// TwinCAT 3 PLC project PowerMonitoringSample
// ProgramVersion: 3.1.4022.3
// libraries:
//   Tc2_Standard, * (Beckhoff Automation GmbH)
//   Tc2_System, * (Beckhoff Automation GmbH)
//   Tc2_Utilities, * (Beckhoff Automation GmbH)
//   Tc3_EventLogger, * (Beckhoff Automation GmbH)
//   Tc3_Module, * (Beckhoff Automation GmbH)
//   Tc3_PowerMonitoring, * (Beckhoff Automation GmbH)
// project tree:
//   DUTs/ E_AnalysisIDs.TcDUT, ST_EL3783_InputSamples.TcDUT, ST_EL3783_InputSamples_Scaled.TcDUT
//   GVLs/ Global_Constants.TcGVL
//   / PlcTask.TcTTO, PlcTaskSlow.TcTTO
//   POUs/ DateTimeClock.TcPOU, MAIN.TcPOU, MAIN_SLOW.TcPOU
//   POUs/TestSignalGeneration/ FB_GenerateInputSignal_1Ph.TcPOU
//   POUs/TestSignalGeneration/SignalGeneration/ E_FunctionType.TcDUT, FB_FunctionGenerator_plusPhi.TcPOU

CONFIGURATION PowerMonitoringSample
    RESOURCE PLC ON TwinCAT3
        TASK PlcTask(INTERVAL := T#1ms, PRIORITY := 4);
        TASK PlcTaskSlow(INTERVAL := T#10ms, PRIORITY := 8);
        PROGRAM MAIN WITH PlcTask : MAIN;
        PROGRAM MAIN_SLOW WITH PlcTaskSlow : MAIN_SLOW;
    END_RESOURCE
END_CONFIGURATION

// ---- DUTs/E_AnalysisIDs.TcDUT
{attribute 'qualified_only'}
{attribute 'strict'}
TYPE E_AnalysisIDs :
(
(* analysis chain TimeBased *)
	 Source_TimeBased :=1,
	 Frequency_TimeBased,
	 BasicValues_TimeBased,
	 PowerValues_TimeBased,
(* analysis chain FrequencyBased *)	
	Source_FrequencyBased,
	PowerValues_FrequencyBased,
	Spectrum_FrequencyBased,
	Harmonics_FrequencyBased	
) UDINT;
END_TYPE

// ---- DUTs/ST_EL3783_InputSamples.TcDUT
TYPE ST_EL3783_InputSamples :
STRUCT
(* Inputs from EL3783 *)
	aUL1		: ARRAY[1..cOversamples] OF INT;
	aUL2		: ARRAY[1..cOversamples] OF INT;
	aUL3		: ARRAY[1..cOversamples] OF INT;
	aIL1		: ARRAY[1..cOversamples] OF INT;
	aIL2		: ARRAY[1..cOversamples] OF INT;
	aIL3		: ARRAY[1..cOversamples] OF INT;
END_STRUCT
END_TYPE

// ---- DUTs/ST_EL3783_InputSamples_Scaled.TcDUT
TYPE ST_EL3783_InputSamples_Scaled :
STRUCT
(* Inputs from EL3783 *)
	aUL1		: ARRAY[1..cOversamples] OF LREAL;
	aUL2		: ARRAY[1..cOversamples] OF LREAL;
	aUL3		: ARRAY[1..cOversamples] OF LREAL;
	aIL1		: ARRAY[1..cOversamples] OF LREAL;
	aIL2		: ARRAY[1..cOversamples] OF LREAL;
	aIL3		: ARRAY[1..cOversamples] OF LREAL;
END_STRUCT
END_TYPE

// ---- POUs/TestSignalGeneration/SignalGeneration/E_FunctionType.TcDUT
TYPE E_FunctionType :
(
	eSine,
	eSquare,
	ePulse,
	eTriangular,
	eSawtooth,	
	eAM
);
END_TYPE

// ---- GVLs/Global_Constants.TcGVL
VAR_GLOBAL CONSTANT
	cOversamples			: UDINT := 10;
	cSamplerate				: UDINT := 10_000;
(*
	cFFTLength				: UDINT := 2048;
	cWindowLength			: UDINT := 1600;	
*)	
	cFFTLength				: UDINT := 4096;
	cWindowLength			: UDINT := 3200;

	cBufferLength			: UDINT := cWindowLength/2;
	
	cHarmonicBands			: UDINT := 20;
	cNumQuantiles			: UDINT := 2;
	cFreqMode				: LREAL := 50.0;
END_VAR

// ---- POUs/MAIN.TcPOU
PROGRAM MAIN
VAR CONSTANT
(* Init parameters*)
	cSourceTimeBasedInitPars		: ST_PMA_Source_InitPars 		   		:= (nBufferLength := cOversamples);	
	cSourceFrequencyBasedInitPars	: ST_PMA_Source_InitPars 		   		:= (nBufferLength := cBufferLength);

	cFrequencyInitPars				: ST_PMA_Frequency_Period_InitPars 		:= (nBufferLength := cOversamples, fSampleRate := cSamplerate, fMinFreq := 40, fMaxFreq := 70, nPeriods := 1, nFilterOrder := 2, fCutoff := 70, eInputSelect := E_PMA_InputSelect.Voltage, fMinInput := 150);
	cBasicValuesInitPars			: ST_PMA_BasicValues_Period_InitPars 	:= (nBufferLength := cOversamples, fSampleRate := cSamplerate, fMinInputCurrent := 0.1);
	cPowerValuesInitPars			: ST_PMA_PowerValues_Period_InitPars 	:= (nBufferLength := cOversamples, fSampleRate := cSamplerate, fMinInputCurrent := 0.1);
	cScalingEL3783Pars				: ST_PMA_Scaling_EL3783_InitPars 	 	:= (nOversamples  := cOversamples, fOffsetVoltage := 0, fGainVoltage := 1, fOffsetCurrent := 0, fGainCurrent := 1, fFactorCurrentTransformer := 1);													
END_VAR
VAR	
(* Inputs*)
	nInputSelect				: INT := 1; 						// 1: generate signal, 2: input EL3783
	stEL3783_1_In 				AT%I* : ST_EL3783_InputSamples;
	stEL3783_1_Scaled			: ST_EL3783_InputSamples_Scaled;
	bEL3783_HcRangeActive 		AT%I* : BOOL;
	aEL3783_HcRange 			AT%I* : ARRAY [0..3] OF USINT;	
	
	fbGenerateInputs			: FB_GenerateInputSignal_1Ph;									
	fSetPhaseDiff				: LREAL := 5;	
	fFreqSetpoint				: LREAL	:= 50;
	fAmplitudeVoltage			: LREAL	:= 230*SQRT(2);
	fAmplitudeCurrent			: LREAL	:= 1*SQRT(2);
	bEnableHarmonics			: BOOL	:= FALSE;

(* Functionblocks *)
	fbScaling					: FB_PMA_Scaling_EL3783 		:= (stInitPars:= cScalingEL3783Pars);
	fbSource_TimeBased			: FB_PMA_Source_1Ph 			:= (nOwnID:= E_AnalysisIDs.Source_TimeBased, 		aDestIDs:= [E_AnalysisIDs.Frequency_TimeBased, E_AnalysisIDs.BasicValues_TimeBased, E_AnalysisIDs.PowerValues_TimeBased], stInitPars:= cSourceTimeBasedInitPars);
	fbSource_FrequencyBased		: FB_PMA_Source_1Ph				:= (nOwnID:= E_AnalysisIDs.Source_FrequencyBased, 	aDestIDs:= [E_AnalysisIDs.PowerValues_FrequencyBased, E_AnalysisIDs.Spectrum_FrequencyBased, E_AnalysisIDs.Harmonics_FrequencyBased], stInitPars:= cSourceFrequencyBasedInitPars);
	fbFrequency					: FB_PMA_Frequency_Period_1Ph 	:= (nOwnID:= E_AnalysisIDs.Frequency_TimeBased, 	stInitPars:= cFrequencyInitPars);
	fbBasicValues				: FB_PMA_BasicValues_Period_1Ph := (nOwnID:= E_AnalysisIDs.BasicValues_TimeBased, 	stInitPars:= cBasicValuesInitPars);
	fbPowerValues				: FB_PMA_PowerValues_Period_1Ph := (nOwnID:= E_AnalysisIDs.PowerValues_TimeBased, 	stInitPars:= cPowerValuesInitPars);
		
(* Control *)
	bResetStatistics			: BOOL;	
	
// Errorhandling
	bError						: BOOL;
	nCountErrors				: UDINT;
	nEventId					: UDINT;
	sEventClassName				: T_MaxString;
	sSourcePath					: T_MaxString;
	eSeverity					: TcEventSeverity;
	ipResultMessage				: I_TcMessage;
	
//Liam's variable for TcHmi
	bResetEnergyRecord : BOOL:= FALSE;
	
END_VAR

bError := FALSE;

(**************************************************************************************************************)
(* Inputs *)
CASE nInputSelect OF
	1:	(* signal generation from PLC *)
		fbGenerateInputs.Call(	bEnableHarmonics			:= bEnableHarmonics,
								fSetFrequency				:= fFreqSetpoint,		// Hz
								fSetAmplitudeVoltage		:= fAmplitudeVoltage,	// peak amplitude of sin signal
								fSetAmplitudeCurrent		:= fAmplitudeCurrent,
								fSetPhasedifferenceCurrent	:= fSetPhaseDiff,
								stEL3783_Scaled				=> stEL3783_1_Scaled);										

	2:	(* signal from terminal *)
		InputEL3783();
		IF fbScaling.bError THEN
			bError := TRUE;
			ipResultMessage := fbScaling.ipResultMessage;
		END_IF
END_CASE

(**************************************************************************************************************)
(* Source *)
fbSource_TimeBased.Call(pBuffer_U:= ADR(stEL3783_1_Scaled.aUL1),			 
						pBuffer_I:= ADR(stEL3783_1_Scaled.aIL1),
						nDataInSizePerCh:= SIZEOF(stEL3783_1_Scaled)/6, // Caused by 3Ph Buffer!
						nOptionPars:= 0);
IF fbSource_TimeBased.bError THEN
	bError := TRUE;
	ipResultMessage := fbSource_TimeBased.ipResultMessage;
END_IF
	
fbSource_FrequencyBased.Call(pBuffer_U:= ADR(stEL3783_1_Scaled.aUL1),			 
							 pBuffer_I:= ADR(stEL3783_1_Scaled.aIL1),		
							 nDataInSizePerCh:= SIZEOF(stEL3783_1_Scaled)/6, // Caused by 3Ph Buffer!
							 nOptionPars:= 0);
IF fbSource_FrequencyBased.bError THEN
	bError := TRUE;
	ipResultMessage := fbSource_FrequencyBased.ipResultMessage;
END_IF
				
(**************************************************************************************************************)
(* Algorithms *)

(* Frequency *)
IF NOT fbFrequency.Call(bResetStatistics:= bResetStatistics) THEN
	bError := TRUE;
	ipResultMessage := fbFrequency.ipResultMessage;	
END_IF

(* Basic Values *)
IF NOT fbBasicValues.Call(fFreq:= fbFrequency.fFreq, bResetStatistics:= bResetStatistics) THEN
	bError := TRUE;
	ipResultMessage := fbBasicValues.ipResultMessage;
END_IF

(* Power Values *)

(*Liam's Code for TcHmi control and Monitor*)
//Thêm biến bResetEnergyRecord vào để điều khiển quá trình reset lại giá trị của kWh
IF NOT fbPowerValues.Call(fFreq:= fbFrequency.fFreq, bResetEnergyCalc := bResetEnergyRecord, bResetStatistics:= bResetStatistics) THEN
	bError := TRUE;
	ipResultMessage := fbPowerValues.ipResultMessage;
END_IF

(**************************************************************************************************************)
(* Event reporting *)
IF ipResultMessage <> 0 THEN	
	nEventId 		:= ipResultMessage.nEventId;
	sSourcePath 	:= ipResultMessage.ipSourceInfo.sName;
	eSeverity 		:= ipResultMessage.eSeverity;
	
	ipResultMessage.RequestEventClassName(1033, sEventClassName, SIZEOF(sEventClassName));
END_IF
IF bError THEN
	nCountErrors := nCountErrors + 1;
END_IF


(*Liam's Code for TcHmi control and Monitor*)
DateTimeClock();

ACTION InputEL3783:
(* //Autorange
fbScaling.Call_1Ph_Autorange(	pInputBuffer_U			:= ADR(stEL3783_1_In.aUL1), 
								pInputBuffer_I			:= ADR(stEL3783_1_In.aIL1), 
								nInputBufferSize		:= SIZEOF(stEL3783_1_In)/6, 
								pOutputBuffer_U			:= ADR(stEL3783_1_Scaled.aUL1), 
								pOutputBuffer_I			:= ADR(stEL3783_1_Scaled.aIL1), 
								nOutputBufferSize		:= SIZEOF(stEL3783_1_Scaled)/6, 
								bEL3783_HcRangeActive	:= bEL3783_HcRangeActive, 
								aEL3783_HcRange			:= aEL3783_HcRange);

*)		
fbScaling.Call_1Ph(	pInputBuffer_U		:= ADR(stEL3783_1_In.aUL1), 
					pInputBuffer_I		:= ADR(stEL3783_1_In.aIL1), 
					nInputBufferSize	:= SIZEOF(stEL3783_1_In)/6, 
					pOutputBuffer_U		:= ADR(stEL3783_1_Scaled.aUL1), 
					pOutputBuffer_I		:= ADR(stEL3783_1_Scaled.aIL1), 
					nOutputBufferSize	:= SIZEOF(stEL3783_1_Scaled)/6,
					bUse_5A_Range		:= FALSE);
END_ACTION

END_PROGRAM

// ---- POUs/TestSignalGeneration/FB_GenerateInputSignal_1Ph.TcPOU
FUNCTION_BLOCK FB_GenerateInputSignal_1Ph
VAR_INPUT
	fSetFrequency						: LREAL:= 50;		// Hz
	fSetAmplitudeVoltage				: LREAL:= 325;		// peak amplitude of sin signal	
	fSetAmplitudeCurrent				: LREAL:= 2;		// peak amplitude of sin signal	
	fSetPhasedifferenceCurrent			: LREAL:= 0;
END_VAR
VAR_OUTPUT
END_VAR
VAR
	fbFunctionGeneratorVoltage_L1_1		: FB_FunctionGenerator_plusPhi;	// Signal generation
	fbFunctionGeneratorVoltage_L1_2		: FB_FunctionGenerator_plusPhi;	// Signal generation
	fbFunctionGeneratorCurrent_L1		: FB_FunctionGenerator_plusPhi;	// Signal generation
	fbFunctionGeneratorCurrent_L1_2		: FB_FunctionGenerator_plusPhi;	// Signal generation
	fbFunctionGeneratorCurrent_L1_3		: FB_FunctionGenerator_plusPhi;	// Signal generation

	aBufferGen_VoltageL1_1				: ARRAY[1..cOversamples] OF LREAL;
	aBufferGen_VoltageL1_2				: ARRAY[1..cOversamples] OF LREAL;
	aBufferGen_CurrentL1_1				: ARRAY[1..cOversamples] OF LREAL;
	aBufferGen_CurrentL1_2				: ARRAY[1..cOversamples] OF LREAL;
	aBufferGen_CurrentL1_3				: ARRAY[1..cOversamples] OF LREAL;
END_VAR

METHOD Call
VAR CONSTANT
	cHarm_U_FreqFactor					: LREAL	:= 20.0; // 20th harmonic
	cHarm_U_AmpFactor					: LREAL	:= 0.1;//0.10;
	
	cHarm_I_FreqFactor_1				: LREAL	:= 7.0;
	cHarm_I_AmpFactor_1					: LREAL	:= 0.015;//0.15;
	cHarm_I_FreqFactor_2				: LREAL	:= 20.0;
	cHarm_I_AmpFactor_2					: LREAL	:= 0.01;//0.10;
END_VAR
VAR_INPUT
	bEnableHarmonics					: BOOL	:= FALSE;
	fSetFrequency						: LREAL	:= 50;		// Hz
	fSetAmplitudeVoltage				: LREAL	:= 325;		// peak amplitude of sin signal	
	fSetAmplitudeCurrent				: LREAL	:= 2;		// peak amplitude of sin signal	
	fSetPhasedifferenceCurrent			: LREAL	:= 0;
END_VAR
VAR_OUTPUT
	stEL3783_Scaled						: ST_EL3783_InputSamples_Scaled;
END_VAR
VAR
	i									: UDINT;
END_VAR
(* signal generator *)		
// L1
fbFunctionGeneratorVoltage_L1_1(fFrequency 	:= fSetFrequency,							// "Voltage - 1st harmonic"
								fAmplitude 	:= fSetAmplitudeVoltage,
								fPhi		:= 0,
								eFunction 	:= E_FunctionType.eSine,
								aSignal		:= aBufferGen_VoltageL1_1);		

fbFunctionGeneratorVoltage_L1_2(fFrequency 	:= fSetFrequency*cHarm_U_FreqFactor,		// "Voltage - harmonic"
								fAmplitude 	:= fSetAmplitudeVoltage*cHarm_U_AmpFactor,
								fPhi		:= 0,
								eFunction 	:= E_FunctionType.eSine,
								aSignal		:= aBufferGen_VoltageL1_2);								

fbFunctionGeneratorCurrent_L1(	fFrequency 	:= fSetFrequency,							// "Current - 1st harmonic"
								fAmplitude 	:= fSetAmplitudeCurrent,
								fPhi		:= -fSetPhasedifferenceCurrent,
								eFunction 	:= E_FunctionType.eSine,
								aSignal		:= aBufferGen_CurrentL1_1);	
								
fbFunctionGeneratorCurrent_L1_2(fFrequency 	:= fSetFrequency*cHarm_I_FreqFactor_1,		// "Voltage - harmonic"
								fAmplitude 	:= fSetAmplitudeCurrent*cHarm_I_AmpFactor_1,
								fPhi		:= (-fSetPhasedifferenceCurrent*cHarm_I_FreqFactor_1),
								eFunction 	:= E_FunctionType.eSine,
								aSignal		:= aBufferGen_CurrentL1_2);			

fbFunctionGeneratorCurrent_L1_3(fFrequency 	:= fSetFrequency*cHarm_I_FreqFactor_2,		// "Voltage - harmonic"
								fAmplitude 	:= fSetAmplitudeCurrent*cHarm_I_AmpFactor_2,
								fPhi		:= (-fSetPhasedifferenceCurrent*cHarm_I_FreqFactor_2),
								eFunction 	:= E_FunctionType.eSine,
								aSignal		:= aBufferGen_CurrentL1_3);									
				
// harmonics
FOR i:=1 TO cOversamples DO	
	IF bEnableHarmonics THEN
		stEL3783_Scaled.aUL1[i] := aBufferGen_VoltageL1_1[i] + aBufferGen_VoltageL1_2[i];
		stEL3783_Scaled.aIL1[i] := aBufferGen_CurrentL1_1[i] + aBufferGen_CurrentL1_2[i] + aBufferGen_CurrentL1_3[i];
	ELSE
		stEL3783_Scaled.aUL1[i] := aBufferGen_VoltageL1_1[i];
		stEL3783_Scaled.aIL1[i] := aBufferGen_CurrentL1_1[i];
	END_IF
END_FOR
END_METHOD

END_FUNCTION_BLOCK

// ---- POUs/TestSignalGeneration/SignalGeneration/FB_FunctionGenerator_plusPhi.TcPOU
// generates a signal build up by the specified function type. v1.2
FUNCTION_BLOCK FB_FunctionGenerator_plusPhi
VAR_INPUT
	bEnable		: BOOL:= TRUE;
	fFrequency	: LREAL:= 1000;	// in [Hz]
	fAmplitude	: LREAL:= 1;
	fPhi		: LREAL	:= 0;		// just for sin / in deg!!
	fOffset		: LREAL;
	nDutyCycle	: UINT:= 50;		// % (for pulse function)
	eFunction	: E_FunctionType:= E_FunctionType.eSine;	
END_VAR
VAR_IN_OUT
	aSignal		: ARRAY[1..10] OF LREAL;	//nOversamples
END_VAR
VAR_OUTPUT
	bError		: BOOL;
END_VAR

VAR
	bInit						: BOOL:= TRUE;
	fbGetTaskIdx				: GETCURTASKINDEX;
	
	fLastFrequency				: LREAL;		// in [Hz]
	fLastAmplitude				: LREAL;
	fLastOffset					: LREAL;
	nLastDutyCycle				: UINT;
	eLastFunction				: E_FunctionType;
	
	nOversamples				: UDINT:= 10;
	
	nSamples					: UDINT;
	fCycleTime					: LREAL;		// in [s]
	fDelta						: LREAL;		// amplitude delta per sample
	fPhase						: LREAL;		// in [°]
	nSign						: INT:= 1;		// 1 or -1
	fLastSignalValue			: LREAL;		// amplitude
	fPeriod						: LREAL;		// in [s]
	fAngularIncrement			: LREAL;		// in [°]
	fAngularIncrementPerCycle	: LREAL;		// in [°]
	fAngularIncrementPerSample	: LREAL;		// in [°]
	(* for modulated signal *)
	fCarrierFrequency			: LREAL:= 500;	// in [Hz] (sine)
	fCarrierAmplitude			: LREAL:= 1;
	fCarrierPeriod				: LREAL;		// in [s]
	fCarrierAngularIncrement			: LREAL;		// in [°]
	fCarrierAngularIncrementPerCycle	: LREAL;		// in [°]
	fCarrierAngularIncrementPerSample	: LREAL;		// in [°]
END_VAR

IF bEnable THEN
	IF fLastFrequency <> fFrequency THEN
		bInit:= TRUE; // For automatic initializing
		fLastFrequency:= fFrequency;
	END_IF
	IF fLastAmplitude <> fAmplitude THEN
		bInit:= TRUE; // For automatic initializing
		fLastAmplitude:= fAmplitude;
	END_IF
	IF fLastOffset <> fOffset THEN
		bInit:= TRUE; // For automatic initializing
		fLastOffset:= fOffset;
	END_IF
	IF nLastDutyCycle <> nDutyCycle THEN
		bInit:= TRUE; // For automatic initializing
		nLastDutyCycle:= nDutyCycle;
	END_IF
	IF eLastFunction <> eFunction THEN
		bInit:= TRUE; // For automatic initializing
		eLastFunction:= eFunction;
	END_IF
	IF bInit THEN
		bError := FALSE;
		// Get taks info	
		fbGetTaskIdx();
		fCycleTime:= TwinCAT_SystemInfoVarList._TaskInfo[fbGetTaskIdx.index].CycleTime (*100ns*) / (10.0 * 1000.0 * 1000.0);	
		fLastSignalValue:= 0;
		nSign:= 1;
		fAngularIncrement:= 0;
		// Flush out old data
		MEMSET(ADR(aSignal), 0, SIZEOF(aSignal));
		IF fFrequency <> 0 AND fCycleTime > 0 THEN
			// Calculate period, increments per plc cycle, increment per oversample
			IF nOversamples <> 0 THEN			
				IF eFunction = E_FunctionType.eSine THEN
					fPeriod:= 1/fFrequency;
					fAngularIncrementPerCycle:= 360*(fCycleTime/fPeriod);
					fAngularIncrementPerSample:= fAngularIncrementPerCycle/nOversamples;
					// no phase adjustment
					bInit:= FALSE;	
				ELSIF eFunction = E_FunctionType.eSquare	THEN
					fPeriod:= 1/fFrequency;
					fAngularIncrementPerCycle:= 360*(fCycleTime/fPeriod);
					fAngularIncrementPerSample:= fAngularIncrementPerCycle/nOversamples;
					fPhase:= 0.5*360;
					bInit:= FALSE;
				ELSIF eFunction = E_FunctionType.ePulse THEN
					fPeriod:= 1/fFrequency;
					fAngularIncrementPerCycle:= 360*(fCycleTime/fPeriod);
					fAngularIncrementPerSample:= fAngularIncrementPerCycle/nOversamples;
					IF nDutyCycle > 100 THEN
						nDutyCycle:= 100;
					END_IF
					fPhase:= (UDINT_TO_LREAL(nDutyCycle)/100)*360;
					bInit:= FALSE;					
				ELSIF eFunction = E_FunctionType.eTriangular THEN
					fPeriod:= 1/fFrequency;				
					fAngularIncrementPerCycle:= 360*(fCycleTime/fPeriod);
					fAngularIncrementPerSample:= fAngularIncrementPerCycle/nOversamples;
					fPhase:= 0.5*360; 
					fDelta:= 4*(fAmplitude/(360/fAngularIncrementPerSample));				
					bInit:= FALSE;
				ELSIF eFunction = E_FunctionType.eSawtooth THEN
					fPeriod:= 1/fFrequency;			
					fAngularIncrementPerCycle:= 360*(fCycleTime/fPeriod);		
					fAngularIncrementPerSample:= fAngularIncrementPerCycle/nOversamples;
					fDelta:= fAmplitude/(360/fAngularIncrementPerSample);
					bInit:= FALSE;
				ELSIF eFunction = E_FunctionType.eAM THEN
					fPeriod:= 1/fFrequency;
					fAngularIncrementPerCycle:= 360*(fCycleTime/fPeriod);
					fAngularIncrementPerSample:= fAngularIncrementPerCycle/nOversamples;
					// no phase adjustment
					fCarrierPeriod:= 1/fCarrierFrequency;
					fCarrierAngularIncrementPerCycle:= 360*(fCycleTime/fCarrierPeriod);
					fCarrierAngularIncrementPerSample:= fCarrierAngularIncrementPerCycle/nOversamples;				
					// no phase adjustment	
					bInit:= FALSE;			
				ELSE
					bError:= TRUE;	
				END_IF
			ELSE
				bError:= TRUE;
			END_IF
		ELSE
			bError:= TRUE;
		END_IF
	END_IF
	
	// Enable function generator
	IF NOT bError THEN		
		CASE eFunction OF		
			// sine: typical for vibrations originating from rotating machine
			E_FunctionType.eSine: Sine();
			
			// square: mixed sine signals good for analyzing spectrum				
			E_FunctionType.eSquare: Square();
			
			// pulse: mixed sine signals good for analyzing spectrum				
			E_FunctionType.ePulse: Pulse();
	
			// sawtooth: ramp-type vibrations, continuously increasing			
			E_FunctionType.eSawtooth: Sawtooth();
		
			// triangular: mixed sine signals good for analyzing spectrum
			E_FunctionType.eTriangular: Triangular();
		
			// amplitude modulation: typical for vibrations originating from gear-tooth failure or bearing faults
			// Carrier signal with own frequency and amplitude		
			E_FunctionType.eAM: AM();			
		END_CASE
	END_IF
ELSE
	// Flush out old data
	MEMSET(ADR(aSignal), 0, SIZEOF(aSignal));
END_IF

METHOD PRIVATE AM
VAR_INPUT
END_VAR
{warning disable C0371}

FOR nSamples:= 1 TO nOversamples DO
	// base signal * carrier signal
	aSignal[nSamples]:= ( fAmplitude*SIN(2*PI*(fAngularIncrement+(nSamples-1)*fAngularIncrementPerSample)/360) + fOffset )
							* ( fCarrierAmplitude*SIN(2*PI*(fCarrierAngularIncrement+(nSamples-1)*fCarrierAngularIncrementPerSample)/360) );
END_FOR
// Increment angular positions
fAngularIncrement:= fAngularIncrement + fAngularIncrementPerCycle;
fCarrierAngularIncrement:= fCarrierAngularIncrement + fCarrierAngularIncrementPerCycle;

{warning restore C0371}
END_METHOD

METHOD PRIVATE Pulse
VAR_INPUT
END_VAR
{warning disable C0371}

FOR nSamples:= 1 TO nOversamples DO
	// For pulse wave (unequal phases)
	IF (fAngularIncrement >= 360) THEN
		fAngularIncrement:= fAngularIncrement - DINT_TO_LREAL(LREAL_TO_DINT(fAngularIncrement/360))*360;
		// or with Tc2_Math library: fAngularIncrement:= LMOD(fAngularIncrement,360);
	END_IF
	IF (fAngularIncrement < fPhase) THEN
		nSign:= 1;		
	ELSIF (fAngularIncrement >= fPhase) THEN
		nSign:= 0;
	END_IF
	fAngularIncrement:= fAngularIncrement + fAngularIncrementPerSample;
	
	aSignal[nSamples]:= nSign*fAmplitude;
	
	aSignal[nSamples]:= aSignal[nSamples] + fOffset;
END_FOR

{warning restore C0371}
END_METHOD

METHOD PRIVATE Sawtooth
VAR_INPUT
END_VAR
{warning disable C0371}

FOR nSamples:= 1 TO nOversamples DO
	// For sawtooth wave (equal phase = period/2)
	IF (fAngularIncrement >= 360) THEN
		fAngularIncrement:= fAngularIncrement - DINT_TO_LREAL(LREAL_TO_DINT(fAngularIncrement/360))*360;
		// or with Tc2_Math library: fAngularIncrement:= LMOD(fAngularIncrement,360);
		fLastSignalValue:= fLastSignalValue -fAmplitude;
	END_IF
	fAngularIncrement:= fAngularIncrement + fAngularIncrementPerSample;

	aSignal[nSamples]:= fLastSignalValue + fDelta;

	// Store last sample
	fLastSignalValue:= aSignal[nSamples];
	
	aSignal[nSamples]:= aSignal[nSamples] + fOffset;					
END_FOR	

{warning restore C0371}
END_METHOD

METHOD PRIVATE Sine
VAR_INPUT
END_VAR
{warning disable C0371}

FOR nSamples:= 1 TO nOversamples DO
	aSignal[nSamples]:= fAmplitude*SIN((2*PI*(fAngularIncrement+(nSamples-1)*fAngularIncrementPerSample)/360)+(fPhi*PI/180)); // sin(x+PhaseDifference) in grad
	aSignal[nSamples]:= aSignal[nSamples] + fOffset;
END_FOR

// Increment angular position
fAngularIncrement:= fAngularIncrement + fAngularIncrementPerCycle;

{warning restore C0371}
END_METHOD

METHOD PRIVATE Square
VAR_INPUT
END_VAR
{warning disable C0371}

FOR nSamples:= 1 TO nOversamples DO
	// For square wave (equal phase = period/2)
	IF (fAngularIncrement >= 360) THEN
		fAngularIncrement:= fAngularIncrement - DINT_TO_LREAL(LREAL_TO_DINT(fAngularIncrement/360))*360;
		// or with Tc2_Math library: fAngularIncrement:= LMOD(fAngularIncrement,360);
	END_IF
	IF (fAngularIncrement < fPhase) THEN
		nSign:= 1;
	ELSIF (fAngularIncrement >= fPhase) THEN
		nSign:= -1;
	END_IF
	fAngularIncrement:= fAngularIncrement + fAngularIncrementPerSample;
	
	aSignal[nSamples]:= nSign*fAmplitude;
	
	aSignal[nSamples]:= aSignal[nSamples] + fOffset;
END_FOR

{warning restore C0371}
END_METHOD

METHOD PRIVATE Triangular
VAR_INPUT
END_VAR
{warning disable C0371}

FOR nSamples:= 1 TO nOversamples DO
	IF (fAngularIncrement >= 360) THEN
		fAngularIncrement:= fAngularIncrement - DINT_TO_LREAL(LREAL_TO_DINT(fAngularIncrement/360))*360;
		// or with Tc2_Math library: fAngularIncrement:= LMOD(fAngularIncrement,360);
	END_IF
	// Negative delta -> Positive delta
	IF fAngularIncrement < fPhase/2 THEN	
		nSign:= 1;		
	ELSIF fAngularIncrement >= fPhase/2 AND fAngularIncrement < 3*fPhase/2 THEN
		nSign:= -1;
	ELSIF fAngularIncrement >= 3*fPhase/2 THEN
		nSign:= 1;	
	END_IF
	fAngularIncrement:= fAngularIncrement + fAngularIncrementPerSample;
	
	aSignal[nSamples]:= fLastSignalValue + nSign*fDelta;
	IF aSignal[nSamples] > fAmplitude THEN
		aSignal[nSamples]:= aSignal[nSamples] - 2*(aSignal[nSamples]-fAmplitude);
	ELSIF aSignal[nSamples] < (-1)*fAmplitude THEN
		aSignal[nSamples]:= aSignal[nSamples] - 2*(aSignal[nSamples]+fAmplitude);
	END_IF
	
	// Store last sample
	fLastSignalValue:= aSignal[nSamples];		
	
	aSignal[nSamples]:= aSignal[nSamples] + fOffset;
END_FOR

{warning restore C0371}
END_METHOD

END_FUNCTION_BLOCK

// ---- POUs/DateTimeClock.TcPOU
PROGRAM DateTimeClock
VAR
	fbSystemTime		: FB_LocalSystemTime;
	dtCurrentDateTime	: DT;
	sCurrentDateTime	: STRING;
	dateDate : DATE;
	todTime : TOD;
	sDate : STRING;
	sTime : STRING;
	fbLow_5m			: TON;
	fbHigh_5m			: TOF;
	pulse5m :BOOL;
	
END_VAR

fbSystemTime(sNetID:='', bEnable:= TRUE, dwCycle:= 5, dwOpt:= 1);	
dtCurrentDateTime	:= SYSTEMTIME_TO_DT(fbSystemTime.systemTime);
sCurrentDateTime	:= MID(DT_TO_STRING(dtCurrentDateTime), 19, 4);
dateDate := DT_TO_DATE(dtCurrentDateTime);
todTime := DT_TO_TOD (dtCurrentDateTime);
sDate := DATE_TO_STRING (dateDate);
sTime := TOD_TO_STRING (todTime);
fbLow_5m(IN			:= NOT pulse5m, PT:= T#1M);
fbHigh_5m(IN		:= fbLow_5m.Q, PT:= T#1M, Q => pulse5m);

END_PROGRAM

// ---- POUs/MAIN_SLOW.TcPOU
PROGRAM MAIN_SLOW
VAR CONSTANT
(* Init parameters *)	
	// FB_PMA_PowerValues																																																				
	cPowerValuesInitPars		: ST_PMA_PowerValues_InitPars:=(fTimeLagCurrentTransformer	:= 0,
																fSampleRate					:= cSamplerate,		// in Hz 
																fBaseFreq					:= cFreqMode,		// in Hz
																nFFT_Length					:= cFFTLength,
																nWindowLength				:= cWindowLength,
																nNumBands					:= cHarmonicBands,
																fBandwidth					:= 20.0,
																eWindowType					:= E_PMA_WindowType.HannWindow);
	// FB_PMA_Spectrum
	cSpectrumInitPars			: ST_PMA_Spectrum_InitPars:=(	nFFT_Length					:= cFFTLength,
																nWindowLength				:= cWindowLength, 
																fSampleRate					:= cSamplerate,		// in Hz
																fDecibelThreshold 			:= GVL_PMA.cMinArgLog10,
																bTransformToDecibel			:= FALSE,             
																eWindowType					:= E_PMA_WindowType.HannWindow,
																eScalingType				:= E_PMA_ScalingType.NoScaling );		
	// FB_PMA_Harmonics										
	cHarmonicsInitPars			: ST_PMA_Harmonics_InitPars:=(	nFFT_Length					:= cFFTLength,
																nWindowLength				:= cWindowLength,
																fSampleRate					:= cSamplerate,		// in Hz
																nNumBands					:= cHarmonicBands,
																fBaseFreq					:= cFreqMode,		// in Hz
																fBandwidth					:= 20.0,
																eWindowType					:= E_PMA_WindowType.HannWindow,	
																bTransformToDecibel			:= FALSE,		
																fDecibelThreshold			:= GVL_PMA.cMinArgLog10,
																bTransformToPercent			:= TRUE);
END_VAR
VAR
(* Functionblocks *)
	fbPowerValues				: FB_PMA_PowerValues_1Ph := (nOwnID:= E_AnalysisIDs.PowerValues_FrequencyBased, stInitPars:= cPowerValuesInitPars);
	fbSpectrum					: FB_PMA_Spectrum_1Ph	 := (nOwnID:= E_AnalysisIDs.Spectrum_FrequencyBased, 	stInitPars:= cSpectrumInitPars);
	fbHarmonics					: FB_PMA_Harmonics_1Ph	 := (nOwnID:= E_AnalysisIDs.Harmonics_FrequencyBased,	stInitPars:= cHarmonicsInitPars);
	
(* Results *)
	// FB_PMA_Spectrum
	aSpectrum					: ARRAY[0..1, 0..cFFTLength/2] OF LREAL;	// dims: (NumPhases*2 | FFTLength/2 + 1)
	// FB_PMA_Harmonics
	aHarmonics					: ARRAY[0..1, 0..cHarmonicBands-1] OF LREAL; // dims: (NumPhases*2 | NumBands)
	
(* Control *)
	bResetStatistics			: BOOL;	
	bResetEnergyCalculation		: BOOL;
	
(* Errorhandling *)
	bError						: BOOL;
	nCountErrors				: UDINT;
	nEventId					: UDINT;
	sEventClassName				: T_MaxString;
	sSourcePath					: T_MaxString;
	eSeverity					: TcEventSeverity;
	ipResultMessage				: I_TcMessage;
END_VAR

bError := FALSE;

(**************************************************************************************************************)
(* Algorithms *)

(* Power Values *)
IF NOT fbPowerValues.Call(	bResetEnergyCalc	:= bResetEnergyCalculation,
							bResetStatistics	:= bResetStatistics)	
THEN
	bError := TRUE;
	ipResultMessage := fbPowerValues.ipResultMessage;
END_IF

(*Spectrum*)
IF NOT fbSpectrum.Call(	ADR(aSpectrum[0,0]), 
						ADR(aSpectrum[1,0]), 
						SIZEOF(aSpectrum)/2)
THEN
	bError := TRUE;
	ipResultMessage := fbSpectrum.ipResultMessage;
END_IF

(* Harmonics *)
IF NOT fbHarmonics.Call(	bResetStatistics	:= bResetStatistics,
							pHarmonicsRMS_U		:= ADR(aHarmonics[0,0]),
							pHarmonicsRMS_I		:= ADR(aHarmonics[1,0]),
							nHarmonicsRMSSize	:= SIZEOF(aHarmonics)/2)
THEN
	bError := TRUE;
	ipResultMessage := fbHarmonics.ipResultMessage;
END_IF

(**************************************************************************************************************)
(* Event reporting *)
IF ipResultMessage <> 0 THEN	
	nEventId 		:= ipResultMessage.nEventId;
	sSourcePath 	:= ipResultMessage.ipSourceInfo.sName;
	eSeverity 		:= ipResultMessage.eSeverity;
	
	ipResultMessage.RequestEventClassName(1033, sEventClassName, SIZEOF(sEventClassName));
END_IF
IF bError THEN
	nCountErrors := nCountErrors + 1;
END_IF

END_PROGRAM
